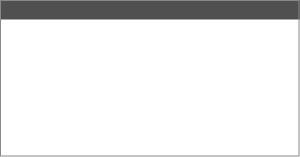
VISUALIZATION CtrlOther  // 300x157
    Rectangle (0,0 300x157)
    Rectangle (0,0 300x19)
END_VISUALIZATION

(* stored: Version 1.1.0.1, ProductVersion 3.1.4024.3
   Visu CtrlOther: Id {7364f4ca-8379-4b93-b42a-6cab8404de00} *)
